// TIA Portal V16 export
// export: Created 2021-09-08T12:46:10.7330699Z, ExportSetting WithDefaults, DisplayName Totally Integrated Automation Portal, DisplayVersion V16 Update 3, DisplayName TIA Portal Version Control Interface, DisplayVersion V16 Update 2, DisplayName TIA Portal Openness, DisplayVersion V16 Update 3, DisplayName TIA Portal Teamcenter Gateway, DisplayVersion V16, DisplayName STEP 7 Professional, DisplayVersion V16 Update 3, DisplayName STEP 7 Safety, DisplayVersion V16, DisplayName WinCC Advanced, DisplayVersion V16 Update 3
FUNCTION_BLOCK "PumpCntr"   // FB60, LAD
{ S7_Optimized_Access := 'FALSE' }
VERSION : 0.1
// #ST:
// номер бита, часло десятичное
//  0  - стоп 
// 0 1 - работа
// 1 2 - запуск
// 2 4 - остановка
// 3 8 - сервисный режим
// 4 16 - ошибка Пуска
// 5 32 - ошибка Стопа
// 6 64 - ошибка питания
// 7 128 - ошибка частотника (дозатора)
// 8 256 - Блокировка внешняя
// 9 - 512 - нажат аварийный стоп
// 10 -1024 - сборная авария
// 11 2048 - местный режим
// 12 4096
// 13 8192
// 14 16384 1-показывать кнопки ручного управления
// 15 32768 - режим 1-ручной, 0-авто (только для индкатора на скаде)
// stored: AutoNumber false, IsIECCheckEnabled false, SetENOAutomatically false, UDAEnableTagReadback false
   VAR_INPUT
      power : Bool;   // питание устройства 1-ок
      run : Bool;   // 1-работа
      emrStop : Bool;   // Авариный стоп 0-авария, 1-ок
      local : Bool;   // 1-местный режим
      alarmFC : Bool;   // 1-авария
      block1 : Bool;
      block2 : Bool;
      block3 : Bool;
      block4 : Bool;
      block5 : Bool;
      block6 : Bool;
      block7 : Bool;
      block8 : Bool;
   END_VAR
   VAR_OUTPUT
      qStart : Bool;   // пуск
   END_VAR
   VAR_IN_OUT
      dev : "Pump";
   END_VAR
   VAR DB_SPECIFIC
      ErrOC : Bool;   // Признак аварии по закрытию или открытию
      ErrPower : Bool;   // Признак аварии питания
      ErrDis : Bool;   // Признак внешней блокировки
      qON : Bool;   // Выход для управления механизмом
      tmrClosing { S7_SetPoint := 'True'} : TON_TIME;
      tmrOpening { S7_SetPoint := 'True'} : TON_TIME;
      closed : Bool;
      opened : Bool;
      closing : Bool;
      opening : Bool;
      errStart : Bool;
      errStop : Bool;
      errEmrStop : Bool;
      errAlarmFc : Bool;
      errService : Bool;
      errLocal : Bool;
      tStart : Time;
      tStop : Time;
   END_VAR
   VAR
      DpumpAckAlarm_Instance : "PumpAckAlarm";
   END_VAR
   VAR CONSTANT
      ACK_DELAY : Time := T#1s;
   END_VAR
BEGIN

REGION Network 1: Сброс состояния
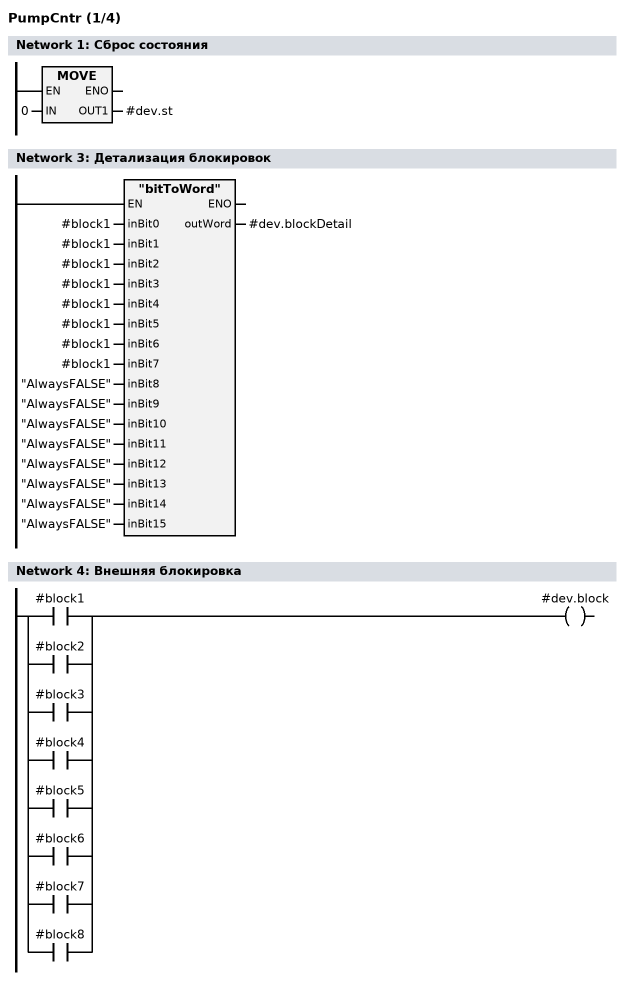
   RUNG wire#powerrail
      { S7_GenerateENO := "TRUE" } Move(in := 0, out1 => #dev.st)
   END_RUNG
   // the same network as SCL:
   #dev.st := 0;
END_REGION

REGION Network 3: Детализация блокировок
   RUNG wire#powerrail
      "bitToWord"(inBit0 := #block1, inBit1 := #block1, inBit2 := #block1, inBit3 := #block1, inBit4 := #block1, inBit5 := #block1, inBit6 := #block1, inBit7 := #block1, inBit8 := "AlwaysFALSE", inBit9 := "AlwaysFALSE", inBit10 := "AlwaysFALSE", inBit11 := "AlwaysFALSE", inBit12 := "AlwaysFALSE", inBit13 := "AlwaysFALSE", inBit14 := "AlwaysFALSE", inBit15 := "AlwaysFALSE", outWord => #dev.blockDetail)
   END_RUNG
   // the same network as SCL:
   "bitToWord"(inBit0 := #block1,
               inBit1 := #block1,
               inBit2 := #block1,
               inBit3 := #block1,
               inBit4 := #block1,
               inBit5 := #block1,
               inBit6 := #block1,
               inBit7 := #block1,
               inBit8 := "AlwaysFALSE",
               inBit9 := "AlwaysFALSE",
               inBit10 := "AlwaysFALSE",
               inBit11 := "AlwaysFALSE",
               inBit12 := "AlwaysFALSE",
               inBit13 := "AlwaysFALSE",
               inBit14 := "AlwaysFALSE",
               inBit15 := "AlwaysFALSE",
               outWord => #dev.blockDetail);
END_REGION

REGION Network 4: Внешняя блокировка
   RUNG wire#powerrail
      Contact( #block1 )
      wire#w1
      Coil( #dev.block )
   END_RUNG
   RUNG wire#powerrail
      Contact( #block2 )
   END_RUNG wire#w1
   RUNG wire#powerrail
      Contact( #block3 )
   END_RUNG wire#w1
   RUNG wire#powerrail
      Contact( #block4 )
   END_RUNG wire#w1
   RUNG wire#powerrail
      Contact( #block5 )
   END_RUNG wire#w1
   RUNG wire#powerrail
      Contact( #block6 )
   END_RUNG wire#w1
   RUNG wire#powerrail
      Contact( #block7 )
   END_RUNG wire#w1
   RUNG wire#powerrail
      Contact( #block8 )
   END_RUNG wire#w1
   // the same network as SCL:
   #dev.block := #block1 OR #block2 OR #block3 OR #block4 OR #block5 OR #block6 OR #block7 OR #block8;
END_REGION

REGION Network 5: Alarms
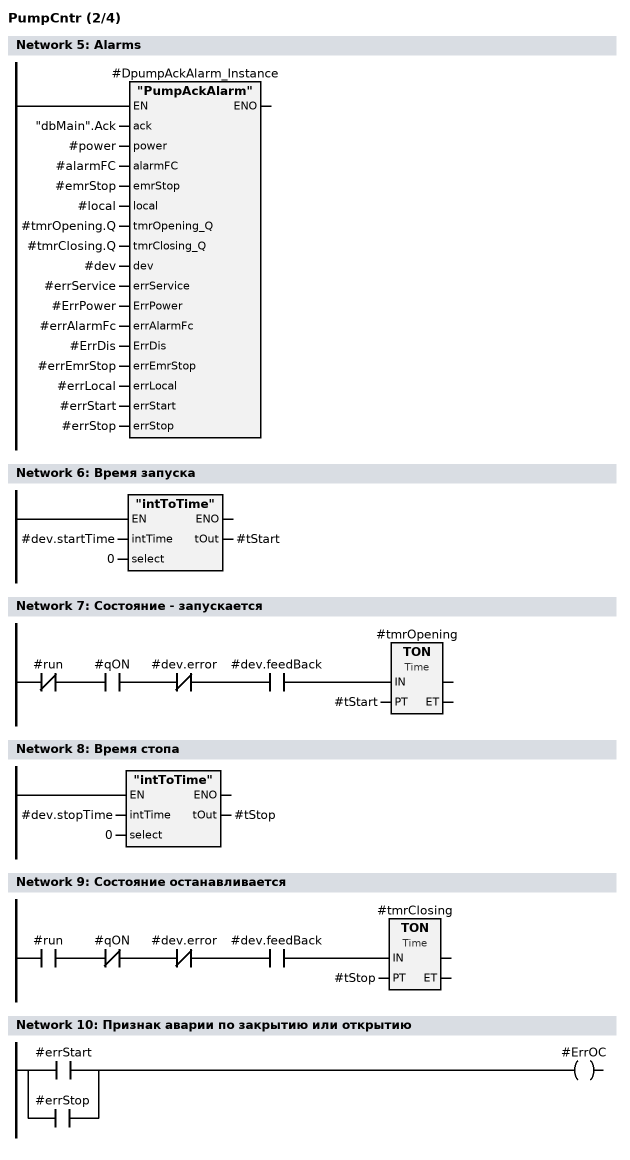
   RUNG wire#powerrail
      #DpumpAckAlarm_Instance(ack := "dbMain".Ack, power := #power, alarmFC := #alarmFC, emrStop := #emrStop, local := #local, tmrOpening_Q := #tmrOpening.Q, tmrClosing_Q := #tmrClosing.Q, dev := #dev, errService := #errService, ErrPower := #ErrPower, errAlarmFc := #errAlarmFc, ErrDis := #ErrDis, errEmrStop := #errEmrStop, errLocal := #errLocal, errStart := #errStart, errStop := #errStop)
   END_RUNG
   // the same network as SCL:
   #DpumpAckAlarm_Instance(ack := "dbMain".Ack,   // "PumpAckAlarm"
                           power := #power,
                           alarmFC := #alarmFC,
                           emrStop := #emrStop,
                           local := #local,
                           tmrOpening_Q := #tmrOpening.Q,
                           tmrClosing_Q := #tmrClosing.Q,
                           dev := #dev,
                           errService := #errService,
                           ErrPower := #ErrPower,
                           errAlarmFc := #errAlarmFc,
                           ErrDis := #ErrDis,
                           errEmrStop := #errEmrStop,
                           errLocal := #errLocal,
                           errStart := #errStart,
                           errStop := #errStop);
END_REGION

REGION Network 6: Время запуска
   RUNG wire#powerrail
      "intToTime"(intTime := #dev.startTime, select := 0, tOut => #tStart)
   END_RUNG
   // the same network as SCL:
   "intToTime"(intTime := #dev.startTime, select := 0, tOut => #tStart);
END_REGION

REGION Network 7: Состояние - запускается
   RUNG wire#powerrail
      I_Contact( #run )
      Contact( #qON )
      I_Contact( #dev.error )
      Contact( #dev.feedBack )
      { S7_Templates := "time_type := Time" } #tmrOpening.TON(pt := #tStart, et =>)
   END_RUNG
   // the same network as SCL:
   #tmrOpening(IN := NOT #run AND #qON AND NOT #dev.error AND #dev.feedBack, PT := #tStart);   // TON
END_REGION

REGION Network 8: Время стопа
   RUNG wire#powerrail
      "intToTime"(intTime := #dev.stopTime, select := 0, tOut => #tStop)
   END_RUNG
   // the same network as SCL:
   "intToTime"(intTime := #dev.stopTime, select := 0, tOut => #tStop);
END_REGION

REGION Network 9: Состояние останавливается
   RUNG wire#powerrail
      Contact( #run )
      I_Contact( #qON )
      I_Contact( #dev.error )
      Contact( #dev.feedBack )
      { S7_Templates := "time_type := Time" } #tmrClosing.TON(pt := #tStop, et =>)
   END_RUNG
   // the same network as SCL:
   #tmrClosing(IN := #run AND NOT #qON AND NOT #dev.error AND #dev.feedBack, PT := #tStop);   // TON
END_REGION

REGION Network 10: Признак аварии по закрытию или открытию
   RUNG wire#powerrail
      Contact( #errStart )
      wire#w1
      Coil( #ErrOC )
   END_RUNG
   RUNG wire#powerrail
      Contact( #errStop )
   END_RUNG wire#w1
   // the same network as SCL:
   #ErrOC := #errStart OR #errStop;
END_REGION

REGION Network 11: Сборная авария
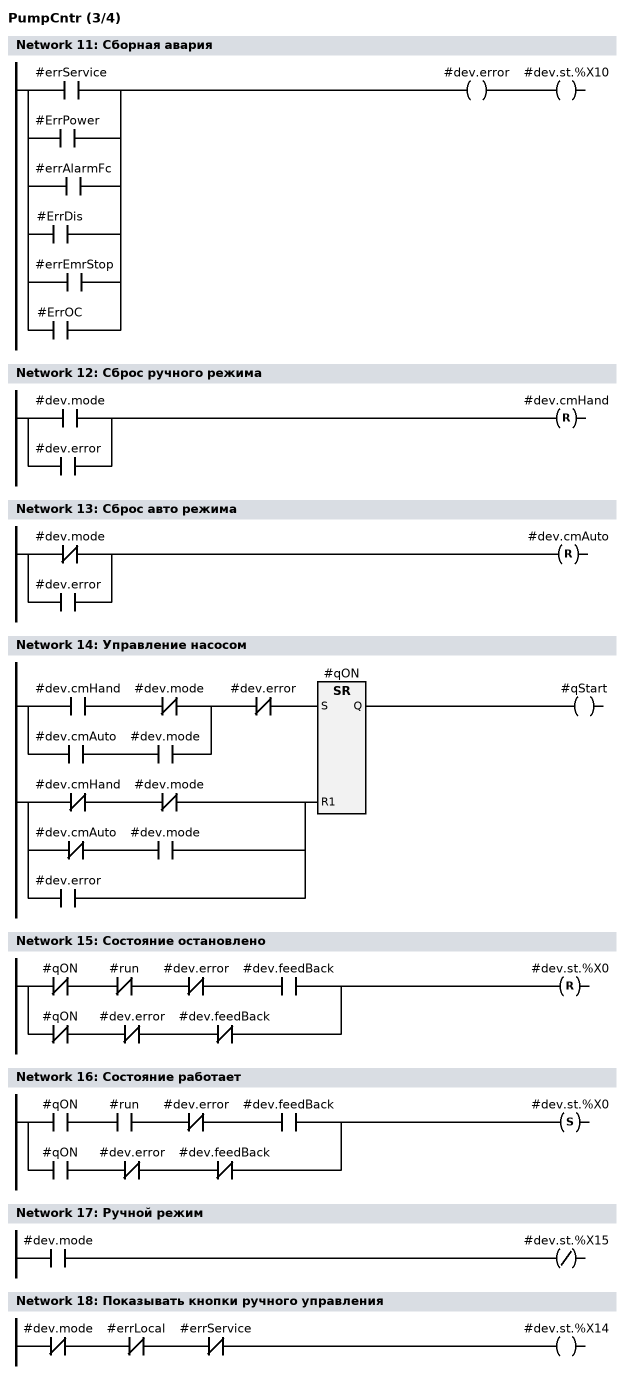
   RUNG wire#powerrail
      Contact( #errService )
      wire#w1
      Coil( #dev.error )
      Coil( #dev.st.%X10 )
   END_RUNG
   RUNG wire#powerrail
      Contact( #ErrPower )
   END_RUNG wire#w1
   RUNG wire#powerrail
      Contact( #errAlarmFc )
   END_RUNG wire#w1
   RUNG wire#powerrail
      Contact( #ErrDis )
   END_RUNG wire#w1
   RUNG wire#powerrail
      Contact( #errEmrStop )
   END_RUNG wire#w1
   RUNG wire#powerrail
      Contact( #ErrOC )
   END_RUNG wire#w1
   // the same network as SCL:
   #dev.error := #errService OR #ErrPower OR #errAlarmFc OR #ErrDis OR #errEmrStop OR #ErrOC;
   #dev.st.%X10 := #dev.error;
END_REGION

REGION Network 12: Сброс ручного режима
   RUNG wire#powerrail
      Contact( #dev.mode )
      wire#w1
      R_Coil( #dev.cmHand )
   END_RUNG
   RUNG wire#powerrail
      Contact( #dev.error )
   END_RUNG wire#w1
   // the same network as SCL:
   IF #dev.mode OR #dev.error THEN #dev.cmHand := FALSE; END_IF;
END_REGION

REGION Network 13: Сброс авто режима
   RUNG wire#powerrail
      I_Contact( #dev.mode )
      wire#w1
      R_Coil( #dev.cmAuto )
   END_RUNG
   RUNG wire#powerrail
      Contact( #dev.error )
   END_RUNG wire#w1
   // the same network as SCL:
   IF NOT #dev.mode OR #dev.error THEN #dev.cmAuto := FALSE; END_IF;
END_REGION

REGION Network 14: Управление насосом
   RUNG wire#powerrail
      Contact( #dev.cmHand )
      I_Contact( #dev.mode )
      wire#w1
      I_Contact( #dev.error )
      S_SR(operand := #qON, r1 := wire#w2)
      Coil( #qStart )
   END_RUNG
   RUNG wire#powerrail
      Contact( #dev.cmAuto )
      Contact( #dev.mode )
   END_RUNG wire#w1
   RUNG wire#powerrail
      I_Contact( #dev.cmHand )
      I_Contact( #dev.mode )
   END_RUNG wire#w2
   RUNG wire#powerrail
      I_Contact( #dev.cmAuto )
      Contact( #dev.mode )
   END_RUNG wire#w2
   RUNG wire#powerrail
      Contact( #dev.error )
   END_RUNG wire#w2
   // the same network as SCL:
   IF ((#dev.cmHand AND NOT #dev.mode) OR (#dev.cmAuto AND #dev.mode)) AND NOT #dev.error THEN
       #qON := TRUE;   // SR flip-flop
   END_IF;
   IF (NOT #dev.cmHand AND NOT #dev.mode) OR (NOT #dev.cmAuto AND #dev.mode) OR #dev.error THEN
       #qON := FALSE;
   END_IF;
   #qStart := #qON;
END_REGION

REGION Network 15: Состояние остановлено
   RUNG wire#powerrail
      I_Contact( #qON )
      I_Contact( #run )
      I_Contact( #dev.error )
      Contact( #dev.feedBack )
      wire#w1
      R_Coil( #dev.st.%X0 )
   END_RUNG
   RUNG wire#powerrail
      I_Contact( #qON )
      I_Contact( #dev.error )
      I_Contact( #dev.feedBack )
   END_RUNG wire#w1
   // the same network as SCL:
   IF (NOT #qON AND NOT #run AND NOT #dev.error AND #dev.feedBack) OR (NOT #qON AND NOT #dev.error AND NOT #dev.feedBack) THEN
       #dev.st.%X0 := FALSE;
   END_IF;
END_REGION

REGION Network 16: Состояние работает
   RUNG wire#powerrail
      Contact( #qON )
      Contact( #run )
      I_Contact( #dev.error )
      Contact( #dev.feedBack )
      wire#w1
      S_Coil( #dev.st.%X0 )
   END_RUNG
   RUNG wire#powerrail
      Contact( #qON )
      I_Contact( #dev.error )
      I_Contact( #dev.feedBack )
   END_RUNG wire#w1
   // the same network as SCL:
   IF (#qON AND #run AND NOT #dev.error AND #dev.feedBack) OR (#qON AND NOT #dev.error AND NOT #dev.feedBack) THEN
       #dev.st.%X0 := TRUE;
   END_IF;
END_REGION

REGION Network 17: Ручной режим
   RUNG wire#powerrail
      Contact( #dev.mode )
      I_Coil( #dev.st.%X15 )
   END_RUNG
   // the same network as SCL:
   #dev.st.%X15 := NOT #dev.mode;
END_REGION

REGION Network 18: Показывать кнопки ручного управления
   RUNG wire#powerrail
      I_Contact( #dev.mode )
      I_Contact( #errLocal )
      I_Contact( #errService )
      Coil( #dev.st.%X14 )
   END_RUNG
   // the same network as SCL:
   #dev.st.%X14 := NOT #dev.mode AND NOT #errLocal AND NOT #errService;
END_REGION

REGION Network 19: Программный выход запуска насоса
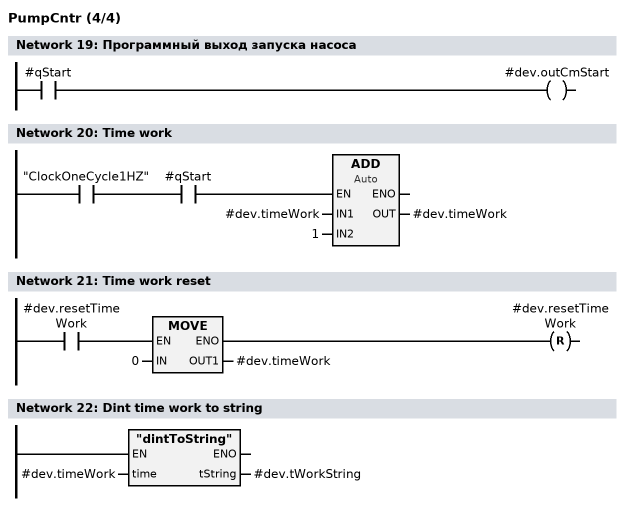
   RUNG wire#powerrail
      Contact( #qStart )
      Coil( #dev.outCmStart )
   END_RUNG
   // the same network as SCL:
   #dev.outCmStart := #qStart;
END_REGION

REGION Network 20: Time work
   RUNG wire#powerrail
      Contact( "ClockOneCycle1HZ" )
      Contact( #qStart )
      Add(in1 := #dev.timeWork, in2 := 1, out => #dev.timeWork)
   END_RUNG
   // the same network as SCL:
   IF "ClockOneCycle1HZ" AND #qStart THEN #dev.timeWork := #dev.timeWork + 1; END_IF;
END_REGION

REGION Network 21: Time work reset
   RUNG wire#powerrail
      Contact( #dev.resetTimeWork )
      Move(in := 0, out1 => #dev.timeWork)
      R_Coil( #dev.resetTimeWork )
   END_RUNG
   // the same network as SCL:
   IF #dev.resetTimeWork THEN
       #dev.timeWork := 0;
       #dev.resetTimeWork := FALSE;
   END_IF;
END_REGION

REGION Network 22: Dint time work to string
   RUNG wire#powerrail
      "dintToString"("time" := #dev.timeWork, tString => #dev.tWorkString)
   END_RUNG
   // the same network as SCL:
   "dintToString"("time" := #dev.timeWork, tString => #dev.tWorkString);
END_REGION
END_FUNCTION_BLOCK
